FUNCTION_BLOCK Test_F_TimeAsString_Returns24HourFormat EXTENDS T_UnitTestBase
VAR
    TimeStruct : TIMESTRUCT := (wHour := 22, wMinute := 20, wSecond := 18);
END_VAR

{attribute 'analysis' := '-33'} // inhibit unused variable warning
METHOD RunTest
IF Retest THEN
	SUPER^.Init();
END_IF

IF TestCompleted THEN
	RETURN;
END_IF

AssertEquals_STRING(Expected := '22:20:18',
                    Actual   := F_TimeAsString(TimeStruct),
                    Message  := 'F_TimeAsString(TimeStruct)');

TestCompleted := TRUE;
END_METHOD

END_FUNCTION_BLOCK

(* stored: Version 1.1.0.1, ProductVersion 3.1.4024.12
   POU Test_F_TimeAsString_Returns24HourFormat: Id {f81aab76-2a34-01f9-2fb5-1c273e9923eb}, SpecialFunc None
   Method RunTest: Id {545b5928-cde2-0810-3770-9f5f2c5f9a7b} *)
